(* CODESYS project BagFeedSequence.Step0_entry.xml

Project tree, tasks and I/O mapping:
*)

// Step0_entry
ACTION Step0_entry:
_attempts := _attempts + 1;
END_ACTION
